TYPE "UDT_ZC_DISP_PPAL_M_VF"
VERSION : 0.1
   STRUCT
      Estado : Bool;   // Estado activado
      SegActivacion : Bool;   // Estado seguridad ok
      Fallo : Bool;   // En fallo
      Orden : Bool;   // Orden activacion
      Consigna : Real := 0.0;   // Consigna
      ValorActual : Real;   // Valor actual
   END_STRUCT;

END_TYPE

